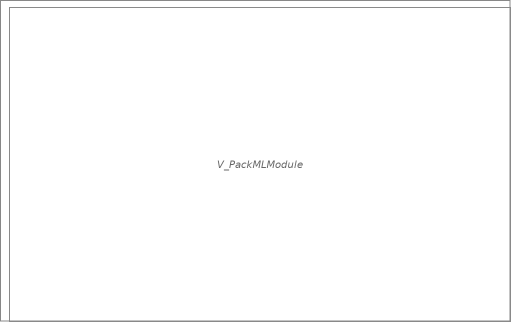
VISUALIZATION V_Main  // 511x322
    Frame (9,7 502x315)
        shows V_PackMLModule(PackML_HMI := MAIN.Machine.Machine_HMI.Statemachine_HMI)
END_VISUALIZATION

(* stored: Version 1.1.0.1, ProductVersion 3.1.4026.18
   Visu V_Main: Id {cd6cf2ea-6909-43c4-8779-52f53bcc55e2} *)
